# EPICS substitutions: elioApp/Db/EL3008.substitutions
file EL3008.template { pattern
{ CHAN	}
{ 1	}
{ 2	}
{ 3	}
{ 4	}
{ 5	}
{ 6	}
{ 7	}
{ 8	}
}
